// TwinCAT 3 PLC project MAS418_PLC
// ProgramVersion: 3.1.4023.0
// libraries:
//   Tc2_Standard, * (Beckhoff Automation GmbH)
//   Tc2_System, * (Beckhoff Automation GmbH)
//   Tc3_Module, * (Beckhoff Automation GmbH)
// project tree:
//   CraneController/FBs/ FB_ClosedLoopControl.TcPOU, FB_MotionRefSelector.TcPOU, FB_OpenLoopControl.TcPOU, FB_StateMachine.TcPOU, FB_MotionRefGenerator.TcPOU, FB_ThetaBoom.TcPOU
//   CraneSimulator/FBs/ FB_CraneSimulator.TcPOU
//   DUTs/ E_Mode.TcDUT, E_Status.TcDUT
//   / GlobalTextList.TcGTLO, PlcTask.TcTTO, Simulator.TcTTO, Visualization Manager.TcVMO (not stored)
//   GVLs/ G_ControllerGreenCrane.TcGVL, G_CylinderState.TcGVL
//   POUs/ MAIN.TcPOU, P_Simulator.TcPOU
//   VISUs/ Visualization.TcVIS
// real-time tasks:
//   TASK PlcTask: cycle T#10ms, priority 20, ADS port 350
//   TASK Simulator: cycle T#100us, priority 1, ADS port 351

CONFIGURATION MAS418_PLC
    RESOURCE PLC ON TwinCAT3
        TASK PlcTask(INTERVAL := T#10ms, PRIORITY := 20);
        TASK Simulator(INTERVAL := T#100us, PRIORITY := 1);
        PROGRAM MAIN WITH PlcTask : MAIN;
        PROGRAM P_Simulator WITH Simulator : P_Simulator;
    END_RESOURCE
END_CONFIGURATION

// ---- DUTs/E_Mode.TcDUT
{attribute 'qualified_only'}
{attribute 'strict'}
TYPE E_Mode :
(
	Manual,
	Auto	
);
END_TYPE

// ---- DUTs/E_Status.TcDUT
{attribute 'qualified_only'}
{attribute 'strict'}
TYPE E_Status :
(
	Ready,
	NotReady,
	Running
);
END_TYPE

// ---- GVLs/G_ControllerGreenCrane.TcGVL
{attribute 'qualified_only'}
VAR_GLOBAL
	bEnable : BOOL;
	bMode : BOOL;
	bStart : BOOL := FALSE;
	bLamp : BOOL := FALSE;
	fVelRef : REAL;
	fTimer : REAL := 0.0;
	eMode : E_Mode;
	eStatus : E_Status;
	fGain : LREAL;
END_VAR

// ---- GVLs/G_CylinderState.TcGVL
{attribute 'qualified_only'}
VAR_GLOBAL
	xm: LREAL;
	ppbar: LREAL;
	prbar: LREAL;
	thetaBoom: LREAL;
END_VAR

// ---- POUs/MAIN.TcPOU
PROGRAM MAIN
VAR
	fbStateMachine : FB_StateMachine;
END_VAR

fbStateMachine();

END_PROGRAM

// ---- CraneController/FBs/FB_StateMachine.TcPOU
FUNCTION_BLOCK FB_StateMachine
VAR_INPUT
END_VAR
VAR_OUTPUT
END_VAR
VAR
	fbMotionSelector : FB_MotionRefSelector;
	fbThetaBoom : FB_ThetaBoom;
END_VAR

IF (G_ControllerGreenCrane.bEnable) THEN
	G_ControllerGreenCrane.eStatus := E_Status.Ready;
	IF (G_ControllerGreenCrane.bMode) THEN
		G_ControllerGreenCrane.eMode := E_Mode.Auto;
		G_ControllerGreenCrane.bLamp := G_ControllerGreenCrane.bStart := FALSE;
	ELSE  
		G_ControllerGreenCrane.eMode := E_Mode.Manual;
		G_ControllerGreenCrane.bLamp := G_ControllerGreenCrane.bStart;
		IF (G_ControllerGreenCrane.bStart) THEN
			G_ControllerGreenCrane.eStatus := E_Status.Running;
		END_IF		
	END_IF
ELSE
	G_ControllerGreenCrane.bStart := G_ControllerGreenCrane.bLamp := FALSE;
	G_ControllerGreenCrane.eStatus := E_Status.NotReady;
	IF (G_ControllerGreenCrane.bMode) THEN
		G_ControllerGreenCrane.eMode := E_Mode.Auto;
	ELSE  
		G_ControllerGreenCrane.eMode := E_Mode.Manual;
	END_IF
END_IF

IF (G_ControllerGreenCrane.bLamp) THEN
	G_ControllerGreenCrane.fTimer := G_ControllerGreenCrane.fTimer + 0.01;
ELSE 
	G_ControllerGreenCrane.fTimer := 0.0;
END_IF


fbMotionSelector(Auto1Man0 := G_ControllerGreenCrane.bMode, xCylRefGenm := 0, vCylRefGenm := 0, vCylJoyms := G_ControllerGreenCrane.fVelRef);
fbThetaBoom(xCylm := G_CylinderState.xm, thetaBoom => G_CylinderState.thetaBoom);

END_FUNCTION_BLOCK

// ---- CraneController/FBs/FB_MotionRefSelector.TcPOU
FUNCTION_BLOCK FB_MotionRefSelector
VAR_INPUT
	Auto1Man0: BOOL;
	xCylRefGenm: LREAL;
	vCylRefGenm: LREAL;
	vCylJoyms: LREAL;
END_VAR
VAR_OUTPUT

END_VAR
VAR
	fbOpenLoopControl : FB_OpenLoopControl;
END_VAR

IF NOT(G_ControllerGreenCrane.eStatus = E_Status.Running) THEN 
	fbOpenLoopControl(bEnable := FALSE, fVelocityReference_ms := vCylJoyms, fMaxValveFlow_lmin := 19, fVelocityFeedForward => G_ControllerGreenCrane.fGain);
ELSIF NOT(Auto1Man0) THEN
    fbOpenLoopControl(bEnable := TRUE, fVelocityReference_ms := vCylJoyms, fMaxValveFlow_lmin := 19, fVelocityFeedForward => G_ControllerGreenCrane.fGain);
ELSE 
	fbOpenLoopControl(bEnable := FALSE, fVelocityReference_ms := vCylJoyms, fMaxValveFlow_lmin := 19, fVelocityFeedForward => G_ControllerGreenCrane.fGain); //This will be Auto
END_IF;

END_FUNCTION_BLOCK

// ---- CraneController/FBs/FB_OpenLoopControl.TcPOU
FUNCTION_BLOCK FB_OpenLoopControl
VAR_INPUT
	bEnable: BOOL;
	fVelocityReference_ms: LREAL;
	fMaxValveFlow_lmin: LREAL;
END_VAR
VAR_OUTPUT
	fVelocityFeedForward: LREAL;
END_VAR
VAR
	rtb_Q_refm3s: LREAL;
END_VAR


(* Outputs for Atomic SubSystem: '<Root>/FB_OpenLoopControl' *)
(* Switch: '<S1>/Switch2' incorporates:
 *  Constant: '<S1>/Annnulus_Area'
 *  Constant: '<S1>/Bore_Area'
 *  Product: '<S1>/Product1'
 *  Product: '<S1>/Product3' *)

IF fVelocityReference_ms >= 0.0 THEN 
    rtb_Q_refm3s := 0.0033183 * fVelocityReference_ms;
ELSE 
    rtb_Q_refm3s := fVelocityReference_ms * 0.0023562;
END_IF;

(* End of Switch: '<S1>/Switch2' *)


(* Switch: '<S1>/Switch1' *)

IF bEnable THEN 
    (* Outport: '<Root>/fVelocityFeedForward' incorporates:
     *  Gain: '<S1>/Gain1'
     *  Product: '<S1>/Divide2' *)
    fVelocityFeedForward := (60000.0 * rtb_Q_refm3s) / fMaxValveFlow_lmin;
ELSE 
    (* Outport: '<Root>/fVelocityFeedForward' incorporates:
     *  Constant: '<S1>/Constant' *)
    fVelocityFeedForward := 0.0;
END_IF;

(* End of Switch: '<S1>/Switch1' *)
(* End of Outputs for SubSystem: '<Root>/FB_OpenLoopControl' *)

END_FUNCTION_BLOCK

// ---- CraneController/FBs/FB_ThetaBoom.TcPOU
FUNCTION_BLOCK FB_ThetaBoom
VAR_INPUT
	xCylm: LREAL;
END_VAR
VAR_OUTPUT
	thetaBoom: LREAL;
END_VAR
VAR
	a: LREAL;
END_VAR


(* MATLAB Function: '<Root>/CylinderDiscplacementToBoomAngle' *)
(* Geomtry Constants *)
(* MATLAB Function 'CylinderDiscplacementToBoomAngle': '<S1>:1' *)
(* '<S1>:1:4' ABx = 0.427; *)
(* '<S1>:1:5' ABy = 1.057; *)
(* '<S1>:1:6' ACx = 0.49484; *)
(* '<S1>:1:7' ACy = 0.133; *)
(* '<S1>:1:9' AB = sqrt(abs(ABx)^2 + abs(ABy)^2); *)
(* '<S1>:1:10' AC = sqrt(abs(ACx)^2 + abs(ACy)^2); *)
(* '<S1>:1:12' BC = 0.77222 + xCyl; *)
(* '<S1>:1:14' alpha1 = atand(abs(ACy)/abs(ACx)); *)
(* '<S1>:1:15' alpha2 = atand(abs(ABy)/abs(ABx)); *)
(* '<S1>:1:17' theta1 = acosd( (abs(AB)^2 + abs(AC)^2 - (abs(BC))^2) / (2 * abs(AB) * abs(AC)) ) - alpha2 + alpha1; *)
a := ABS(xCylm + 0.77222);
(* Outport: '<Root>/thetaBoom' incorporates:
 *  MATLAB Function: '<Root>/CylinderDiscplacementToBoomAngle' *)
(* '<S1>:1:19' thetaBoom = theta1; *)
thetaBoom := ((ACOS((1.5621336256 - (a * a)) / 1.1682662621269122) * 57.295779513082323) - 68.00259659335785) + 15.044069585156381;

END_FUNCTION_BLOCK

// ---- POUs/P_Simulator.TcPOU
PROGRAM P_Simulator
VAR
	fbCraneSimulator : FB_CraneSimulator;
END_VAR

IF (G_ControllerGreenCrane.fTimer = 0.0) THEN 
	fbCraneSimulator(ssMethodType := 0, uDCV := G_ControllerGreenCrane.fGain, xm => G_CylinderState.xm, ppbar => G_CylinderState.ppbar, prbar => G_CylinderState.prbar);
ELSE 
	fbCraneSimulator(ssMethodType := 1, uDCV := G_ControllerGreenCrane.fGain, xm => G_CylinderState.xm, ppbar => G_CylinderState.ppbar, prbar => G_CylinderState.prbar);
END_IF

END_PROGRAM

// ---- CraneSimulator/FBs/FB_CraneSimulator.TcPOU
FUNCTION_BLOCK FB_CraneSimulator
VAR_INPUT
	ssMethodType: SINT;
	uDCV: LREAL;
END_VAR
VAR_OUTPUT
	xm: LREAL;
	ppbar: LREAL;
	prbar: LREAL;
END_VAR
VAR
	pLS: LREAL;
	QDCV_in: LREAL;
	rtb_xDot: LREAL;
	y: LREAL;
	temp1: LREAL;
	temp2: LREAL;
	temp3: LREAL;
	temp4: LREAL;
	c_DiscreteTimeIntegrator_DS: LREAL;
	c_DiscreteTimeIntegrator1_D: LREAL;
	c_DiscreteTimeIntegrator2_D: LREAL;
	c_DiscreteTimeIntegrator3_D: LREAL;
END_VAR



CASE ssMethodType OF
    0: 
        (* SystemInitialize for Atomic SubSystem: '<Root>/CraneSimulator' *)
        (* InitializeConditions for DiscreteIntegrator: '<S1>/Discrete-Time Integrator' *)
        c_DiscreteTimeIntegrator_DS := 0.0;
        (* InitializeConditions for DiscreteIntegrator: '<S1>/Discrete-Time Integrator1' *)
        c_DiscreteTimeIntegrator1_D := 0.0;
        (* InitializeConditions for DiscreteIntegrator: '<S1>/Discrete-Time Integrator2' *)
        c_DiscreteTimeIntegrator2_D := 4.377E+6;
        (* InitializeConditions for DiscreteIntegrator: '<S1>/Discrete-Time Integrator3' *)
        c_DiscreteTimeIntegrator3_D := 468300.0;
        (* End of SystemInitialize for SubSystem: '<Root>/CraneSimulator' *)
    1: 
        (* Outputs for Atomic SubSystem: '<Root>/CraneSimulator' *)
        (* DiscreteIntegrator: '<S1>/Discrete-Time Integrator' *)
        rtb_xDot := c_DiscreteTimeIntegrator_DS;
        (* Outport: '<Root>/x [m]' incorporates:
         *  DiscreteIntegrator: '<S1>/Discrete-Time Integrator1' *)
        xm := c_DiscreteTimeIntegrator1_D;
        (* Outport: '<Root>/pp [bar]' incorporates:
         *  DiscreteIntegrator: '<S1>/Discrete-Time Integrator2'
         *  Gain: '<S1>/Gain' *)
        ppbar := 1.0E-5 * c_DiscreteTimeIntegrator2_D;
        (* Outport: '<Root>/pr [bar]' incorporates:
         *  DiscreteIntegrator: '<S1>/Discrete-Time Integrator3'
         *  Gain: '<S1>/Gain1' *)
        prbar := 1.0E-5 * c_DiscreteTimeIntegrator3_D;
        (* MATLAB Function: '<S1>/MATLAB Function' incorporates:
         *  DiscreteIntegrator: '<S1>/Discrete-Time Integrator'
         *  DiscreteIntegrator: '<S1>/Discrete-Time Integrator1'
         *  DiscreteIntegrator: '<S1>/Discrete-Time Integrator2'
         *  DiscreteIntegrator: '<S1>/Discrete-Time Integrator3' *)
        (* Parameters *)
        (* MATLAB Function 'CraneSimulator/MATLAB Function': '<S2>:1' *)
        (* '<S2>:1:3' Fexternal = 1.3365e+04; *)
        (* [N] *)
        (* '<S2>:1:4' mEffective = 1.3365e+04; *)
        (* [kg] *)
        (* '<S2>:1:5' kFric = 4000; *)
        (* [N/(ms)] *)
        (* '<S2>:1:6' Apiston = 0.0033; *)
        (* [m^2] *)
        (* '<S2>:1:7' Aannulus = 0.0023; *)
        (* [m^2] *)
        (* '<S2>:1:8' beta = 1.0e9; *)
        (* [Pa] *)
        (* '<S2>:1:9' pSupply = 180e5; *)
        (* [Pa] *)
        (* '<S2>:1:10' pReturn = 1.1e5; *)
        (* [Pa] *)
        (* '<S2>:1:11' MaxStroke = 0.5; *)
        (* [m] *)
        (* '<S2>:1:12' VCyl_A = 1.0e-03; *)
        (* '<S2>:1:13' VCyl_B = 1.25e-03; *)
        (* '<S2>:1:14' p_nom_DCV = 7e5; *)
        (* '<S2>:1:15' Q1_ref_DCV = 20/6e4; *)
        (* '<S2>:1:16' kv1_DCV = Q1_ref_DCV/sqrt(p_nom_DCV); *)
        (* '<S2>:1:17' p0 = 7e5; *)
        (* compensator crack pressure *)
        (* Directional Control Valve - Lifting Cylinder  *)
        (* LS Pressure *)
        (* '<S2>:1:20' if uDCV > 0 *)

        IF uDCV > 0.0 THEN 
            (* '<S2>:1:21' pLS = pPiston; *)
            pLS := c_DiscreteTimeIntegrator2_D;
        ELSIF uDCV < 0.0 THEN 
            (* '<S2>:1:22' elseif uDCV < 0 *)
            (* '<S2>:1:23' pLS = pRod; *)
            pLS := c_DiscreteTimeIntegrator3_D;
        ELSE 
            (* '<S2>:1:24' else *)
            (* '<S2>:1:25' pLS = 0; *)
            pLS := 0.0;
        END_IF;

        (* '<S2>:1:28' if pLS<0 *)

        IF pLS < 0.0 THEN 
            (* '<S2>:1:29' pLS = 0; *)
            pLS := 0.0;
        END_IF;

        (* Pressure Compensator *)
        (* '<S2>:1:33' pPC = 0; *)
        (* '<S2>:1:35' if p0 <= (pSupply - pLS) *)

        IF (1.8E+7 - pLS) >= 700000.0 THEN 
            (* '<S2>:1:36' pPC = pLS+p0; *)
            pLS := pLS + 700000.0;
        ELSE 
            (* '<S2>:1:37' elseif 0 < (pSupply - pLS) < p0 *)
            (* '<S2>:1:38' pPC = pSupply-pLS; *)
            pLS := 1.8E+7 - pLS;
        END_IF;

        (* '<S2>:1:43' if pPC<0 *)

        IF pLS < 0.0 THEN 
            (* '<S2>:1:44' pPC = 0; *)
            pLS := 0.0;
        END_IF;

        (* Orifice Equations *)
        (* '<S2>:1:47' if uDCV > 0 *)

        IF uDCV > 0.0 THEN 
            (* '<S2>:1:48' QDCV_in =  kv1_DCV*uDCV*sign(pPC-pPiston)*sqrt(abs(pPC-pPiston)); *)
            pLS := pLS - c_DiscreteTimeIntegrator2_D;

            IF pLS < 0.0 THEN 
                y := -1.0;
            ELSIF pLS > 0.0 THEN 
                y := 1.0;
            ELSE 
                y := 0.0;
            END_IF;

            temp3 := ABS(pLS);
            QDCV_in := ((3.9840953644479785E-7 * uDCV) * y) * SQRT(temp3);
            (* '<S2>:1:49' QDCV_out = kv1_DCV*uDCV*sign(pRod-pReturn)*sqrt(abs(pRod-pReturn)); *)

            IF (c_DiscreteTimeIntegrator3_D - 110000.0) < 0.0 THEN 
                y := -1.0;
            ELSIF (c_DiscreteTimeIntegrator3_D - 110000.0) > 0.0 THEN 
                y := 1.0;
            ELSE 
                y := 0.0;
            END_IF;

            temp4 := ABS(c_DiscreteTimeIntegrator3_D - 110000.0);
            pLS := ((3.9840953644479785E-7 * uDCV) * y) * SQRT(temp4);
        ELSIF uDCV < 0.0 THEN 
            (* '<S2>:1:50' elseif uDCV < 0 *)
            (* '<S2>:1:51' QDCV_out =  kv1_DCV*uDCV*sign(pPC-pRod)*sqrt(abs(pPC-pRod)); *)
            pLS := pLS - c_DiscreteTimeIntegrator3_D;

            IF pLS < 0.0 THEN 
                y := -1.0;
            ELSIF pLS > 0.0 THEN 
                y := 1.0;
            ELSE 
                y := 0.0;
            END_IF;

            temp1 := ABS(pLS);
            pLS := ((3.9840953644479785E-7 * uDCV) * y) * SQRT(temp1);
            (* '<S2>:1:52' QDCV_in =  kv1_DCV*uDCV*sign(pRod-pReturn)*sqrt(abs(pRod-pReturn)); *)

            IF (c_DiscreteTimeIntegrator3_D - 110000.0) < 0.0 THEN 
                y := -1.0;
            ELSIF (c_DiscreteTimeIntegrator3_D - 110000.0) > 0.0 THEN 
                y := 1.0;
            ELSE 
                y := 0.0;
            END_IF;

            temp2 := ABS(c_DiscreteTimeIntegrator3_D - 110000.0);
            QDCV_in := ((3.9840953644479785E-7 * uDCV) * y) * SQRT(temp2);
        ELSE 
            (* '<S2>:1:53' else *)
            (* '<S2>:1:54' QDCV_in = 0; *)
            QDCV_in := 0.0;
            (* '<S2>:1:55' QDCV_out = 0; *)
            pLS := 0.0;
        END_IF;

        (* Pressure Gradients *)
        (* '<S2>:1:58' VA = VCyl_A + x*Apiston; *)
        (* '<S2>:1:59' VB =  VCyl_B + (MaxStroke - x)*Aannulus; *)
        (* '<S2>:1:60' VA_dot = Apiston*xDot; *)
        (* '<S2>:1:61' VB_dot = -Aannulus*xDot; *)
        (* '<S2>:1:62' pPistonDot = beta/VA*(QDCV_in - VA_dot); *)
        QDCV_in := (1.0E+9 / ((c_DiscreteTimeIntegrator1_D * 0.0033) + 0.001)) * (QDCV_in - (0.0033 * c_DiscreteTimeIntegrator_DS));
        (* '<S2>:1:63' pRodDot = beta/VB*(-QDCV_out - VB_dot); *)
        pLS := (1.0E+9 / (((0.5 - c_DiscreteTimeIntegrator1_D) * 0.0023) + 0.00125)) * (( -pLS) - (-0.0023 * c_DiscreteTimeIntegrator_DS));
        (* Update for DiscreteIntegrator: '<S1>/Discrete-Time Integrator' incorporates:
         *  DiscreteIntegrator: '<S1>/Discrete-Time Integrator2'
         *  DiscreteIntegrator: '<S1>/Discrete-Time Integrator3'
         *  MATLAB Function: '<S1>/MATLAB Function' *)
        (* Viscouse Friction *)
        (* '<S2>:1:66' Ffric = kFric*xDot; *)
        (* Hydraulic Force *)
        (* '<S2>:1:69' Fhyd = pPiston*Apiston - pRod*Aannulus; *)
        (* Newton Second Law of Motion *)
        (* '<S2>:1:72' xDotDot = (Fhyd - Ffric - Fexternal)/mEffective; *)
        c_DiscreteTimeIntegrator_DS := ((((((c_DiscreteTimeIntegrator2_D * 0.0033) - (c_DiscreteTimeIntegrator3_D * 0.0023)) - (4000.0 * c_DiscreteTimeIntegrator_DS)) - 13365.0) / 13365.0) * 0.0001) + c_DiscreteTimeIntegrator_DS;

        IF c_DiscreteTimeIntegrator_DS >= 0.12 THEN 
            c_DiscreteTimeIntegrator_DS := 0.12;
        ELSIF c_DiscreteTimeIntegrator_DS <= -0.12 THEN 
            c_DiscreteTimeIntegrator_DS := -0.12;
        END_IF;

        (* End of Update for DiscreteIntegrator: '<S1>/Discrete-Time Integrator' *)
        

        (* Update for DiscreteIntegrator: '<S1>/Discrete-Time Integrator1' *)
        c_DiscreteTimeIntegrator1_D := (0.0001 * rtb_xDot) + c_DiscreteTimeIntegrator1_D;

        IF c_DiscreteTimeIntegrator1_D >= 0.5 THEN 
            c_DiscreteTimeIntegrator1_D := 0.5;
        ELSIF c_DiscreteTimeIntegrator1_D <= 0.0 THEN 
            c_DiscreteTimeIntegrator1_D := 0.0;
        END_IF;

        (* End of Update for DiscreteIntegrator: '<S1>/Discrete-Time Integrator1' *)
        

        (* Update for DiscreteIntegrator: '<S1>/Discrete-Time Integrator2' *)
        c_DiscreteTimeIntegrator2_D := (0.0001 * QDCV_in) + c_DiscreteTimeIntegrator2_D;

        IF c_DiscreteTimeIntegrator2_D >= 1.8E+7 THEN 
            c_DiscreteTimeIntegrator2_D := 1.8E+7;
        ELSIF c_DiscreteTimeIntegrator2_D <= 110000.0 THEN 
            c_DiscreteTimeIntegrator2_D := 110000.0;
        END_IF;

        (* End of Update for DiscreteIntegrator: '<S1>/Discrete-Time Integrator2' *)
        

        (* Update for DiscreteIntegrator: '<S1>/Discrete-Time Integrator3' *)
        c_DiscreteTimeIntegrator3_D := (0.0001 * pLS) + c_DiscreteTimeIntegrator3_D;

        IF c_DiscreteTimeIntegrator3_D >= 1.8E+7 THEN 
            c_DiscreteTimeIntegrator3_D := 1.8E+7;
        ELSIF c_DiscreteTimeIntegrator3_D <= 110000.0 THEN 
            c_DiscreteTimeIntegrator3_D := 110000.0;
        END_IF;

        (* End of Update for DiscreteIntegrator: '<S1>/Discrete-Time Integrator3' *)
        (* End of Outputs for SubSystem: '<Root>/CraneSimulator' *)
END_CASE;

END_FUNCTION_BLOCK

// ---- CraneController/FBs/FB_ClosedLoopControl.TcPOU
FUNCTION_BLOCK FB_ClosedLoopControl
VAR_INPUT
	ssMethodType: SINT;
	bEnable: BOOL;
	bActivateIntegralController: BOOL;
	fProportionalGain: LREAL;
	fIntegralGain: LREAL;
	fPositionReference: LREAL;
	fPositionFeedback: LREAL;
	bIntegralControllReset: BOOL;
END_VAR
VAR_OUTPUT
	fClosedLoopPosition: LREAL;
	fPositionError: LREAL;
END_VAR
VAR
	rtb_u_FB: LREAL;
	rtb_Saturation1: LREAL;
	c_DiscreteTimeIntegrator_DS: LREAL;
END_VAR



CASE ssMethodType OF
    0: 
        (* SystemInitialize for Atomic SubSystem: '<Root>/FB_ClosedLoopControl' *)
        (* InitializeConditions for DiscreteIntegrator: '<S1>/Discrete-Time Integrator' *)
        c_DiscreteTimeIntegrator_DS := 0.0;
        (* End of SystemInitialize for SubSystem: '<Root>/FB_ClosedLoopControl' *)
    1: 
        (* Outputs for Atomic SubSystem: '<Root>/FB_ClosedLoopControl' *)
        (* Sum: '<S1>/Sum1' *)
        fPositionError := fPositionReference - fPositionFeedback;
        (* DiscreteIntegrator: '<S1>/Discrete-Time Integrator' *)

        IF bIntegralControllReset THEN 
            c_DiscreteTimeIntegrator_DS := 0.0;
        END_IF;


        IF c_DiscreteTimeIntegrator_DS >= 1.0 THEN 
            c_DiscreteTimeIntegrator_DS := 1.0;
        ELSIF c_DiscreteTimeIntegrator_DS <= -1.0 THEN 
            c_DiscreteTimeIntegrator_DS := -1.0;
        END_IF;

        (* Switch: '<S1>/Switch' incorporates:
         *  Constant: '<S1>/Constant'
         *  DiscreteIntegrator: '<S1>/Discrete-Time Integrator' *)

        IF bActivateIntegralController THEN 
            rtb_u_FB := c_DiscreteTimeIntegrator_DS;
        ELSE 
            rtb_u_FB := 0.0;
        END_IF;

        (* End of Switch: '<S1>/Switch' *)
        

        (* Sum: '<S1>/Sum5' incorporates:
         *  Product: '<S1>/Product' *)
        rtb_u_FB := (fProportionalGain * fPositionError) + rtb_u_FB;
        (* Saturate: '<S1>/Saturation1' *)

        IF rtb_u_FB > 1.0 THEN 
            rtb_Saturation1 := 1.0;
        ELSIF rtb_u_FB >= -1.0 THEN 
            rtb_Saturation1 := rtb_u_FB;
        ELSE 
            rtb_Saturation1 := -1.0;
        END_IF;

        (* End of Saturate: '<S1>/Saturation1' *)
        

        (* Switch: '<S1>/Switch1' *)

        IF bEnable THEN 
            (* Outport: '<Root>/fClosedLoopPosition' *)
            fClosedLoopPosition := rtb_Saturation1;
        ELSE 
            (* Outport: '<Root>/fClosedLoopPosition' incorporates:
             *  Constant: '<S1>/Constant1' *)
            fClosedLoopPosition := 0.0;
        END_IF;

        (* End of Switch: '<S1>/Switch1' *)
        

        (* Update for DiscreteIntegrator: '<S1>/Discrete-Time Integrator' incorporates:
         *  Product: '<S1>/Divide'
         *  Product: '<S1>/Product2'
         *  Sum: '<S1>/Sum2'
         *  Sum: '<S1>/Sum3' *)
        c_DiscreteTimeIntegrator_DS := (((((rtb_Saturation1 - rtb_u_FB) / fProportionalGain) + fPositionError) * fIntegralGain) * 0.01) + c_DiscreteTimeIntegrator_DS;

        IF c_DiscreteTimeIntegrator_DS >= 1.0 THEN 
            c_DiscreteTimeIntegrator_DS := 1.0;
        ELSIF c_DiscreteTimeIntegrator_DS <= -1.0 THEN 
            c_DiscreteTimeIntegrator_DS := -1.0;
        END_IF;

        (* End of Update for DiscreteIntegrator: '<S1>/Discrete-Time Integrator' *)
        (* End of Outputs for SubSystem: '<Root>/FB_ClosedLoopControl' *)
END_CASE;

END_FUNCTION_BLOCK

// ---- CraneController/FBs/FB_MotionRefGenerator.TcPOU
FUNCTION_BLOCK FB_MotionRefGenerator
VAR_INPUT
	Enable: BOOL;
	x0m: LREAL;
	v0ms: LREAL;
	Position_SPm: LREAL;
	Velocity_SPms: LREAL;
	t0s: LREAL;
	tRamps: LREAL;
	tHoldPoss: LREAL;
	SimulationTimes: LREAL;
END_VAR
VAR_OUTPUT
	PositionRefm: LREAL;
	VelocityRefms: LREAL;
END_VAR
VAR
	Error: DINT;
	slopeExt: LREAL;
	tHold: LREAL;
	x1: LREAL;
	x4: LREAL;
	rtb_Saturation3: LREAL;
	x1_tmp: LREAL;
	x1_tmp_tmp: LREAL;
	x4_tmp: LREAL;
	x4_tmp_tmp: LREAL;
	x4_tmp_tmp_0: LREAL;
	x1_tmp_0: LREAL;
END_VAR


(* Outputs for Atomic SubSystem: '<Root>/RampMotionProfileGenerator' *)
(* Saturate: '<S1>/Saturation3' *)

IF Position_SPm > 0.5 THEN 
    rtb_Saturation3 := 0.5;
ELSIF Position_SPm >= 0.0 THEN 
    rtb_Saturation3 := Position_SPm;
ELSE 
    rtb_Saturation3 := 0.0;
END_IF;

(* End of Saturate: '<S1>/Saturation3' *)


(* Saturate: '<S1>/Saturation2' *)

IF Velocity_SPms > 0.12 THEN 
    PositionRefm := 0.12;
ELSIF Velocity_SPms >= 0.0 THEN 
    PositionRefm := Velocity_SPms;
ELSE 
    PositionRefm := 0.0;
END_IF;

(* End of Saturate: '<S1>/Saturation2' *)


(* MATLAB Function: '<S1>/RampSignal' *)
(* MATLAB Function 'RampMotionProfileGenerator/RampSignal': '<S2>:1' *)
(* '<S2>:1:2' x_SP = x_ref - x0; *)
(* '<S2>:1:3' vs=v_ref; *)
(* '<S2>:1:4' slopeExt=v0-vs; *)
slopeExt := v0ms - PositionRefm;
(* '<S2>:1:5' slopeRetr=-vs-v0; *)
(* '<S2>:1:7' as = vs/tRamp; *)
(* '<S2>:1:8' s_acc=(vs^2-v0^2)/as; *)
(* '<S2>:1:10' tHold=(x_SP-s_acc)/vs; *)
tHold := ((rtb_Saturation3 - x0m) - (((PositionRefm * PositionRefm) - (v0ms * v0ms)) / (PositionRefm / tRamps))) / PositionRefm;
(* '<S2>:1:12' if tHold < 0 *)

IF tHold < 0.0 THEN 
    (* '<S2>:1:13' Error = 1; *)
    Error := 1;
ELSE 
    (* '<S2>:1:14' else *)
    (* '<S2>:1:15' Error = 0; *)
    Error := 0;
END_IF;

(* '<S2>:1:18' t1=tRamp; *)
(* '<S2>:1:19' t2=tHold; *)
(* '<S2>:1:20' t3=tRamp; *)
(* '<S2>:1:21' t4=tWait; *)
(* '<S2>:1:22' t5=t1; *)
(* '<S2>:1:23' t6=t2; *)
(* '<S2>:1:24' t7=t3; *)
(* '<S2>:1:26' x1 = x0 + v0*((t0+t1)-t0)-(slopeExt/t1)*((t0+t1)-t0)^2/2; *)
x1_tmp_tmp := t0s + tRamps;
x1_tmp := x1_tmp_tmp - t0s;
x1_tmp_0 := slopeExt / tRamps;
x1 := ((x1_tmp * v0ms) + x0m) - ((x1_tmp_0 * (x1_tmp * x1_tmp)) / 2.0);
(* '<S2>:1:27' x2 = x1 + vs*((t0+t1+t2)-(t0+t1)); *)
(* '<S2>:1:28' x4 = x_ref - v0*((t0+t1+t2+t3+t4+t5)-(t0+t1+t2+t3+t4))+(slopeRetr/t5)*((t0+t1+t2+t3+t4+t5)-(t0+t1+t2+t3+t4))^2/2; *)
x4_tmp_tmp := x1_tmp_tmp + tHold;
x4_tmp_tmp_0 := x4_tmp_tmp + tRamps;
x4_tmp := x4_tmp_tmp_0 + tHoldPoss;
x4 := (x4_tmp + tRamps) - x4_tmp;
x1_tmp := (( -PositionRefm) - v0ms) / tRamps;
x4 := (rtb_Saturation3 - (x4 * v0ms)) + ((x1_tmp * (x4 * x4)) / 2.0);
(* '<S2>:1:29' x5 = x4-vs*((t0+t1+t2+t3+t4+t5+t6)-(t0+t1+t2+t3+t4+t5)); *)
(* '<S2>:1:31' if Error == 1 *)

IF Error = 1 THEN 
    (* '<S2>:1:32' x = x0; *)
    rtb_Saturation3 := x0m;
    (* '<S2>:1:33' v = v0; *)
    PositionRefm := v0ms;
ELSIF (SimulationTimes >= 0.0) AND (SimulationTimes < t0s) THEN 
    (* '<S2>:1:34' elseif t>=0 && t<t0 *)
    (* '<S2>:1:35' x = x0; *)
    rtb_Saturation3 := x0m;
    (* '<S2>:1:36' v = v0; *)
    PositionRefm := v0ms;
ELSIF (SimulationTimes >= t0s) AND (SimulationTimes < x1_tmp_tmp) THEN 
    (* '<S2>:1:37' elseif t>=t0 && t<(t0+t1) *)
    (* '<S2>:1:38' x = x0 + v0*(t-t0)-(slopeExt/t1)*(t-t0)^2/2; *)
    x1_tmp := SimulationTimes - t0s;
    rtb_Saturation3 := ((x1_tmp * v0ms) + x0m) - ((x1_tmp_0 * (x1_tmp * x1_tmp)) / 2.0);
    (* '<S2>:1:39' v = v0-(slopeExt/t1)*(t-t0); *)
    PositionRefm := v0ms - (x1_tmp_0 * x1_tmp);
ELSIF (SimulationTimes >= x1_tmp_tmp) AND (SimulationTimes < x4_tmp_tmp) THEN 
    (* '<S2>:1:40' elseif t>=(t0+t1) && t<(t0+t1+t2) *)
    (* '<S2>:1:41' x = x1 + vs*(t-(t0+t1)); *)
    rtb_Saturation3 := ((SimulationTimes - x1_tmp_tmp) * PositionRefm) + x1;
    (* '<S2>:1:42' v = vs; *)
ELSIF (SimulationTimes >= x4_tmp_tmp) AND (SimulationTimes < x4_tmp_tmp_0) THEN 
    (* '<S2>:1:43' elseif t>=(t0+t1+t2) && t<(t0+t1+t2+t3) *)
    (* '<S2>:1:44' x = x2+vs*(t-(t0+t1+t2))+(slopeExt/t3)*(t-(t0+t1+t2))^2/2; *)
    tHold := (t0s + tRamps) + tHold;
    x1_tmp := SimulationTimes - tHold;
    rtb_Saturation3 := ((((tHold - x1_tmp_tmp) * PositionRefm) + x1) + (x1_tmp * PositionRefm)) + ((x1_tmp_0 * (x1_tmp * x1_tmp)) / 2.0);
    (* '<S2>:1:45' v = vs+(slopeExt/t3)*(t-(t0+t1+t2)); *)
    PositionRefm := (x1_tmp * (slopeExt / tRamps)) + PositionRefm;
ELSIF (SimulationTimes >= x4_tmp_tmp_0) AND (SimulationTimes < x4_tmp) THEN 
    (* '<S2>:1:46' elseif t>=(t0+t1+t2+t3) && t<(t0+t1+t2+t3+t4) *)
    (* '<S2>:1:47' x = x_ref; *)
    (* '<S2>:1:48' v = v0; *)
    PositionRefm := v0ms;
ELSE 
    x1_tmp_0 := ((x1_tmp_tmp + tHold) + tRamps) + tHoldPoss;
    slopeExt := x1_tmp_0 + tRamps;

    IF (SimulationTimes >= x1_tmp_0) AND (SimulationTimes < slopeExt) THEN 
        (* '<S2>:1:49' elseif t>=(t0+t1+t2+t3+t4) && t<(t0+t1+t2+t3+t4+t5) *)
        (* '<S2>:1:50' x = x_ref - v0*(t-(t0+t1+t2+t3+t4))+(slopeRetr/t5)*(t-(t0+t1+t2+t3+t4))^2/2; *)
        x1_tmp_0 := SimulationTimes - x1_tmp_0;
        rtb_Saturation3 := (rtb_Saturation3 - (x1_tmp_0 * v0ms)) + ((x1_tmp * (x1_tmp_0 * x1_tmp_0)) / 2.0);
        (* '<S2>:1:51' v = v0+(slopeRetr/t5)*(t-(t0+t1+t2+t3+t4)); *)
        PositionRefm := (x1_tmp_0 * x1_tmp) + v0ms;
    ELSE 
        x1_tmp_0 := slopeExt + tHold;

        IF (SimulationTimes >= slopeExt) AND (SimulationTimes < x1_tmp_0) THEN 
            (* '<S2>:1:52' elseif t>=(t0+t1+t2+t3+t4+t5) && t<(t0+t1+t2+t3+t4+t5+t6) *)
            (* '<S2>:1:53' x = x4-vs*(t-(t0+t1+t2+t3+t4+t5)); *)
            rtb_Saturation3 := x4 - ((SimulationTimes - slopeExt) * PositionRefm);
            (* '<S2>:1:54' v = -vs; *)
            PositionRefm :=  -PositionRefm;
        ELSIF (SimulationTimes >= x1_tmp_0) AND (SimulationTimes < (x1_tmp_0 + tRamps)) THEN 
            (* '<S2>:1:55' elseif t>=(t0+t1+t2+t3+t4+t5+t6) && t<(t0+t1+t2+t3+t4+t5+t6+t7) *)
            (* '<S2>:1:56' x = x5-vs*(t-(t0+t1+t2+t3+t4+t5+t6))-(slopeRetr/t3)*(t-(t0+t1+t2+t3+t4+t5+t6))^2/2; *)
            tHold := SimulationTimes - x1_tmp_0;
            rtb_Saturation3 := ((x4 - ((x1_tmp_0 - slopeExt) * PositionRefm)) - (tHold * PositionRefm)) - ((x1_tmp * (tHold * tHold)) / 2.0);
            (* '<S2>:1:57' v = -vs-(slopeRetr/t3)*(t-(t0+t1+t2+t3+t4+t5+t6)); *)
            PositionRefm := ( -PositionRefm) - (tHold * x1_tmp);
        ELSE 
            (* '<S2>:1:58' else *)
            (* '<S2>:1:59' x = x0; *)
            rtb_Saturation3 := x0m;
            (* '<S2>:1:60' v = v0; *)
            PositionRefm := v0ms;
        END_IF;

    END_IF;

END_IF;

(* End of MATLAB Function: '<S1>/RampSignal' *)


(* Switch: '<S1>/Switch' *)
(* '<S2>:1:63' T = t0+t1+t2+t3+t4+t5+t6+t7; *)

IF  NOT Enable THEN 
    PositionRefm := v0ms;
END_IF;

(* End of Switch: '<S1>/Switch' *)


(* Saturate: '<S1>/Saturation' *)

IF PositionRefm > 150.0 THEN 
    (* Outport: '<Root>/VelocityRef [m//s]' *)
    VelocityRefms := 150.0;
ELSIF PositionRefm >= -150.0 THEN 
    (* Outport: '<Root>/VelocityRef [m//s]' *)
    VelocityRefms := PositionRefm;
ELSE 
    (* Outport: '<Root>/VelocityRef [m//s]' *)
    VelocityRefms := -150.0;
END_IF;

(* End of Saturate: '<S1>/Saturation' *)


(* Switch: '<S1>/Switch1' *)

IF Enable THEN 
    PositionRefm := rtb_Saturation3;
ELSE 
    PositionRefm := x0m;
END_IF;

(* End of Switch: '<S1>/Switch1' *)


(* Saturate: '<S1>/Saturation1' *)

IF PositionRefm > 500.0 THEN 
    (* Outport: '<Root>/PositionRef [m] ' *)
    PositionRefm := 500.0;
ELSIF PositionRefm < 0.0 THEN 
    (* Outport: '<Root>/PositionRef [m] ' *)
    PositionRefm := 0.0;
END_IF;

(* End of Saturate: '<S1>/Saturation1' *)
(* End of Outputs for SubSystem: '<Root>/RampMotionProfileGenerator' *)

END_FUNCTION_BLOCK

// ---- GlobalTextList.TcGTLO
TEXTLIST GlobalTextList
  62 = '%0.001f'
  602 = '%0.01f'
  556 = '%0.11f'
  529 = '%0.1f'
  399 = '%0.2f'
  262 = '%d'
  559 = '%f'
  221 = '%f,2'
  766 = '%i'
  679 = '100% accurate Angle, (smart match here)'
  591 = 'Auto'
  675 = 'Boom Angle: %0.1f [deg]'
  130 = 'ControlGreenCrane'
  500 = 'ControllerGreenCrane'
  350 = 'Cylinder Position: %f  [m/s]'
  494 = 'Cylinder Position: %f  [m]'
  186 = 'Cylinder Velocity Reference:'
  639 = 'Cylinder Velocity: %f  [m/s]'
  28 = 'Enable'
  670 = 'GroupBox'
  287 = 'Manual'
  791 = 'Mode : %s'
  252 = 'Mode: %s'
  280 = 'ppBar: %0.1f'
  67 = 'ppBar: %0.1f\tprBar: %0.1f'
  927 = 'ppBar: %0.1f [bar]'
  96 = 'prBar: %0.1f [bar]'
  39 = 'Running'
  807 = 'Start'
  311 = 'Status: %s'
  687 = 'Time: %0.1f [s]'
END_TEXTLIST

// ---- VISUs/Visualization.TcVIS
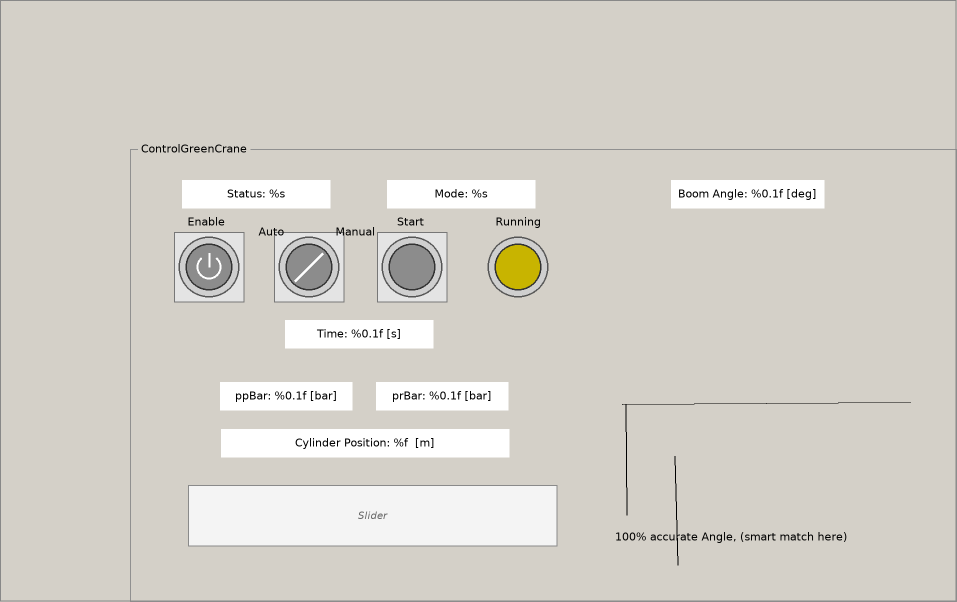
VISUALIZATION Visualization  // 957x602
    GroupBox (130,141 827x461), "ControlGreenCrane"
        Slider (58,344 369x61), variable: G_ControllerGreenCrane.fVelRef, scale -0.12..0.12
        PowerSwitch (44,91 70x70), variable: G_ControllerGreenCrane.bEnable, behaviour: TOGGLE, style: Switch-PowerSwitch-Gray
        RotarySwitch (144,91 70x70), variable: G_ControllerGreenCrane.bMode, behaviour: TOGGLE, style: Switch-RotarySwitch-Gray
        PushSwitch (247,91 70x70), variable: G_ControllerGreenCrane.bStart, behaviour: TOGGLE, style: Switch-PushSwitch-Gray
        Lamp1 (353,91 70x70), variable: G_ControllerGreenCrane.bLamp, style: Lamp-Lamp1-Yellow
        Textfield (51,38 150x30), "Status: %s", text variable: G_ControllerGreenCrane.eStatus
        Textfield (256,38 150x30), "Mode: %s", text variable: G_ControllerGreenCrane.eMode
        Textfield (90,287 290x30), "Cylinder Position: %f [m]", text variable: G_CylinderState.xm
        Textfield (89,240 134x30), "ppBar: %0.1f [bar]", text variable: G_CylinderState.ppbar
        Textfield (154,178 150x30), "Time: %0.1f [s]", text variable: G_ControllerGreenCrane.fTimer
        Label (90,80 103x22), "Auto"
        Label (337,70 103x22), "Running"
        Label (229,70 103x22), "Start"
        Label (25,70 103x22), "Enable"
        Label (174,80 103x22), "Manual"
        Textfield (245,240 134x30), "prBar: %0.1f [bar]", text variable: G_CylinderState.prbar
        Textfield (540,38 155x30), "Boom Angle: %0.1f [deg]", text variable: G_CylinderState.thetaBoom
        Line (492,263) (780,261)
            p2277200375: G_CylinderState.thetaBoom
            p874137650: -288+288*cos(G_CylinderState.thetaBoom*2*3.14/360)
            p1126004900: -288*sin(G_CylinderState.thetaBoom*2*3.14/360)
        Line (497,374) (496,263)
        Line (548,424) (545,315)
        Label (473,381 257x30), "100% accurate Angle, (smart match here)"
END_VISUALIZATION
